PROGRAM MAIN
VAR
	MotorControl : FB_MotorControl;
END_VAR

MotorControl( button1 := GVL_IO.Button1,
	          button2 := GVL_IO.Button2,
	          sensor := GVL_IO.Sensor,
			  Motor => GVL_IO.Motor);

END_PROGRAM

(* stored: Version 1.1.0.1, ProductVersion 3.1.4024.12
   POU MAIN: Id {8af06183-f6c7-4a59-b72a-18871108f6e8}, SpecialFunc None *)
